(* PLC project test.project, CODESYS CODESYS V3.5 SP16 Patch 1 *)
(* stored: creationDateTime 2026-07-09T16:28:26.4121321, modificationDateTime 2026-07-09T16:27:49.6262181 *)

PROGRAM TEST
  VAR
    A : REAL;
    TON1 : TON;
  END_VAR
  VAR  (* added by the conversion: wires and edge detectors of the diagram *)
    _ADD11_OUT : ANY;
    _GE3_OUT : BOOL;
    _SEL18_OUT : BOOL;
  END_VAR

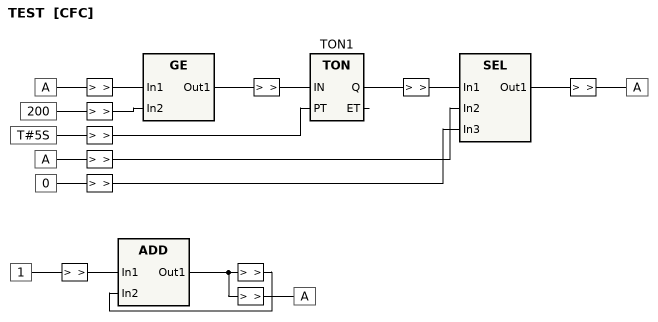
(* CFC diagram, written out as Structured Text *)
_ADD11_OUT := 1 + _ADD11_OUT;
A := _ADD11_OUT;
_GE3_OUT := A >= 200;
TON1(IN := _GE3_OUT, PT := T#5S);
_SEL18_OUT := SEL(TON1.Q, A, 0);
A := _SEL18_OUT;
END_PROGRAM

PROGRAM PLC_PRG

                    TEST();

                  
END_PROGRAM

CONFIGURATION Device
  RESOURCE Application ON PLC
    TASK MainTask(INTERVAL := T#500ms, PRIORITY := 1);
    PROGRAM PLC_PRG WITH MainTask : PLC_PRG;
  END_RESOURCE
END_CONFIGURATION
